// Mitsubishi GX Works2 project: 0709-더블터치   PLC: Q02/Q02H

PROGRAM MAIN
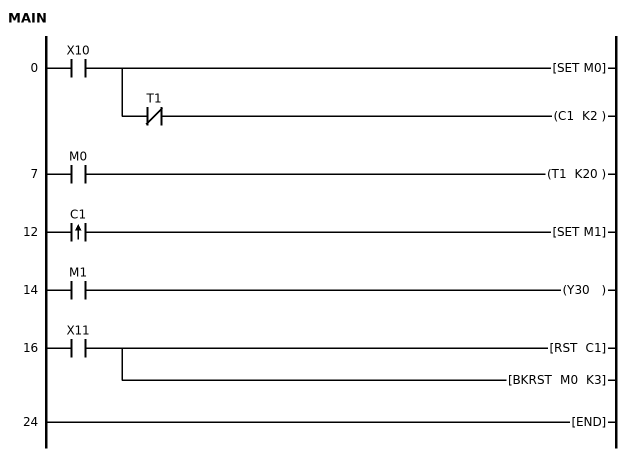
0     LD      X10
      SET     M0
      ANI     T1
      OUT     C1 K2
7     LD      M0
      OUT     T1 K20
12    LDP     C1
      SET     M1
14    LD      M1
      OUT     Y30
16    LD      X11
      RST     C1
      BKRST   M0 K3
24    END
END_PROGRAM
